LIN {X 0,Y 207.14,Z 939.529,A -85,B 0,C 180,E1 3943.742,E2 3943.742} C_VEL
LIN {X 0,Y 198.487,Z 955.966,A -85,B 0,C 180,E1 3942.665,E2 3942.665} C_VEL
LIN {X 0,Y 188.51,Z 971.483,A -85,B 0,C 180,E1 3941.219,E2 3941.219} C_VEL
LIN {X 0,Y 181.932,Z 980.299,A -85,B 0,C 180,E1 3940.126,E2 3940.126} C_VEL
LIN {X 0,Y 176.912,Z 986.053,A -85,B 0,C 180,E1 3939.583,E2 3939.583} C_VEL
LIN {X 0,Y 163.761,Z 998.092,A -85,B 0,C 180,E1 3939.087,E2 3939.087} C_VEL
LIN {X 0,Y 158.072,Z 1003.016,A -85,B 0,C 180,E1 3938.449,E2 3938.449} C_VEL
LIN {X 0,Y 156.561,Z 1004.358,A -85,B 0,C 180,E1 3938.141,E2 3938.141} C_VEL
LIN {X 0,Y 143.715,Z 1015.358,A -85,B 0,C 180,E1 3934.746,E2 3934.746} C_VEL
LIN {X 0,Y 130.308,Z 1025.353,A -85,B 0,C 180,E1 3930.116,E2 3930.116} C_VEL
LIN {X 0,Y 117.407,Z 1033.723,A -85,B 0,C 180,E1 3924,E2 3924} C_VEL
LIN {X 0,Y 106.333,Z 1040.15,A -85,B 0,C 180,E1 3916.387,E2 3916.387} C_VEL
LIN {X 0,Y 97.29,Z 1045.033,A -85,B 0,C 180,E1 3906.587,E2 3906.587} C_VEL
LIN {X 0,Y 91.724,Z 1048.097,A -85,B 0,C 180,E1 3895.157,E2 3895.157} C_VEL
LIN {X 0,Y 90.099,Z 1049.373,A -85,B 0,C 180,E1 3882.822,E2 3882.822} C_VEL
LIN {X 0,Y 91.754,Z 1048.914,A -85,B 0,C 180,E1 3871.872,E2 3871.872} C_VEL
LIN {X 0,Y 92.174,Z 1048.688,A -85,B 0,C 180,E1 3869.998,E2 3869.998} C_VEL
LIN {X 0,Y 90.722,Z 1045.5,A -85,B 0,C 180,E1 3859.842,E2 3859.842} C_VEL
LIN {X 0,Y 91.315,Z 1042.059,A -85,B 0,C 180,E1 3851.484,E2 3851.484} C_VEL
LIN {X 0,Y 94.601,Z 1042.585,A -85,B 0,C 180,E1 3838.807,E2 3838.807} C_VEL
LIN {X 0,Y 102.981,Z 1041.2,A -85,B 0,C 180,E1 3827.182,E2 3827.182} C_VEL
LIN {X 0,Y 114.76,Z 1038.132,A -85,B 0,C 180,E1 3818.213,E2 3818.213} C_VEL
LIN {X 0,Y 128.946,Z 1033.447,A -85,B 0,C 180,E1 3811.464,E2 3811.464} C_VEL
LIN {X 0,Y 142.861,Z 1028.016,A -85,B 0,C 180,E1 3806.958,E2 3806.958} C_VEL
LIN {X 0,Y 130.089,Z 1030.018,A -85,B 0,C 180,E1 3802.123,E2 3802.123} C_VEL
LIN {X 0,Y 117.737,Z 1030.209,A -85,B 0,C 180,E1 3795.768,E2 3795.768} C_VEL
LIN {X 0,Y 107.836,Z 1028.587,A -85,B 0,C 180,E1 3788.53,E2 3788.53} C_VEL
LIN {X 0,Y 99.584,Z 1024.866,A -85,B 0,C 180,E1 3779.424,E2 3779.424} C_VEL
LIN {X 0,Y 94.46,Z 1019.527,A -85,B 0,C 180,E1 3769.876,E2 3769.876} C_VEL
LIN {X 0,Y 91.911,Z 1012.221,A -85,B 0,C 180,E1 3759.627,E2 3759.627} C_VEL
LIN {X 0,Y 91.679,Z 1004.049,A -85,B 0,C 180,E1 3750.607,E2 3750.607} C_VEL
LIN {X 0,Y 93.237,Z 993.607,A -85,B 0,C 180,E1 3741.524,E2 3741.524} C_VEL
LIN {X 0,Y 95.373,Z 985.119,A -85,B 0,C 180,E1 3735.378,E2 3735.378} C_VEL
LIN {X 0,Y 97.55,Z 984.863,A -85,B 0,C 180,E1 3732.439,E2 3732.439} C_VEL
LIN {X 0,Y 100.039,Z 984.278,A -85,B 0,C 180,E1 3730.517,E2 3730.517} C_VEL
LIN {X 0,Y 103.465,Z 983.965,A -85,B 0,C 180,E1 3727.585,E2 3727.585} C_VEL
LIN {X 0,Y 106.11,Z 983.483,A -85,B 0,C 180,E1 3725.867,E2 3725.867} C_VEL
LIN {X 0,Y 110.9,Z 982.693,A -85,B 0,C 180,E1 3723.018,E2 3723.018} C_VEL
LIN {X 0,Y 118.293,Z 981.361,A -85,B 0,C 180,E1 3719.47,E2 3719.47} C_VEL
LIN {X 0,Y 120.142,Z 980.967,A -85,B 0,C 180,E1 3718.741,E2 3718.741} C_VEL
LIN {X 0,Y 112.253,Z 991.51,A -85,B 0,C 180,E1 3713.075,E2 3713.075} C_VEL
LIN {X 0,Y 104.884,Z 1000.824,A -85,B 0,C 180,E1 3706.05,E2 3706.05} C_VEL
LIN {X 0,Y 98.718,Z 1008.666,A -85,B 0,C 180,E1 3697.568,E2 3697.568} C_VEL
LIN {X 0,Y 94.402,Z 1015.031,A -85,B 0,C 180,E1 3687.573,E2 3687.573} C_VEL
LIN {X 0,Y 92.584,Z 1019.589,A -85,B 0,C 180,E1 3676.894,E2 3676.894} C_VEL
LIN {X 0,Y 93.405,Z 1022.419,A -85,B 0,C 180,E1 3666,E2 3666} C_VEL
LIN {X 0,Y 96.968,Z 1023.539,A -85,B 0,C 180,E1 3655.453,E2 3655.453} C_VEL
LIN {X 0,Y 103.213,Z 1022.966,A -85,B 0,C 180,E1 3645.776,E2 3645.776} C_VEL
LIN {X 0,Y 111.857,Z 1020.637,A -85,B 0,C 180,E1 3637.295,E2 3637.295} C_VEL
LIN {X 0,Y 122.487,Z 1016.449,A -85,B 0,C 180,E1 3630.088,E2 3630.088} C_VEL
LIN {X 0,Y 133.914,Z 1010.597,A -85,B 0,C 180,E1 3624.372,E2 3624.372} C_VEL
LIN {X 0,Y 145.608,Z 1003.273,A -85,B 0,C 180,E1 3619.825,E2 3619.825} C_VEL
LIN {X 0,Y 158.047,Z 993.888,A -85,B 0,C 180,E1 3615.932,E2 3615.932} C_VEL
LIN {X 0,Y 169.51,Z 983.568,A -85,B 0,C 180,E1 3612.953,E2 3612.953} C_VEL
LIN {X 0,Y 180.948,Z 971.298,A -85,B 0,C 180,E1 3610.405,E2 3610.405} C_VEL
LIN {X 0,Y 191.03,Z 958.248,A -85,B 0,C 180,E1 3608.419,E2 3608.419} C_VEL
LIN {X 0,Y 200.358,Z 943.599,A -85,B 0,C 180,E1 3606.749,E2 3606.749} C_VEL
LIN {X 0,Y 208.396,Z 927.988,A -85,B 0,C 180,E1 3605.407,E2 3605.407} C_VEL
LIN {X 0,Y 214.864,Z 911.992,A -85,B 0,C 180,E1 3604.36,E2 3604.36} C_VEL
LIN {X 0,Y 220.066,Z 894.686,A -85,B 0,C 180,E1 3603.504,E2 3603.504} C_VEL
LIN {X 0,Y 223.579,Z 876.803,A -85,B 0,C 180,E1 3602.869,E2 3602.869} C_VEL
LIN {X 0,Y 229.364,Z 828.556,A -85,B 0,C 180,E1 3601.817,E2 3601.817} C_VEL
LIN {X 0,Y 228.68,Z 825.976,A -85,B 0,C 180,E1 3598.998,E2 3598.998} C_VEL
LIN {X 0,Y 228.398,Z 824.641,A -85,B 0,C 180,E1 3595.481,E2 3595.481} C_VEL
LIN {X 0,Y 228.531,Z 825.221,A -85,B 0,C 180,E1 3592.964,E2 3592.964} C_VEL
LIN {X 0,Y 229.196,Z 827.412,A -85,B 0,C 180,E1 3589.824,E2 3589.824} C_VEL
LIN {X 0,Y 229.508,Z 828.787,A -85,B 0,C 180,E1 3588.784,E2 3588.784} C_VEL
LIN {X 0,Y 222.463,Z 886.283,A -85,B 0,C 180,E1 3587.683,E2 3587.683} C_VEL
LIN {X 0,Y 218.345,Z 904.811,A -85,B 0,C 180,E1 3587.221,E2 3587.221} C_VEL
LIN {X 0,Y 212.708,Z 922.213,A -85,B 0,C 180,E1 3586.66,E2 3586.66} C_VEL
LIN {X 0,Y 205.625,Z 938.773,A -85,B 0,C 180,E1 3585.946,E2 3585.946} C_VEL
LIN {X 0,Y 196.716,Z 955.353,A -85,B 0,C 180,E1 3584.953,E2 3584.953} C_VEL
LIN {X 0,Y 186.536,Z 970.767,A -85,B 0,C 180,E1 3583.628,E2 3583.628} C_VEL
LIN {X 0,Y 175.18,Z 985.129,A -85,B 0,C 180,E1 3581.861,E2 3581.861} C_VEL
LIN {X 0,Y 162.615,Z 998.588,A -85,B 0,C 180,E1 3579.484,E2 3579.484} C_VEL
LIN {X 0,Y 156.561,Z 1004.358,A -85,B 0,C 180,E1 3578.141,E2 3578.141} C_VEL
LIN {X 0,Y 150.863,Z 1009.035,A -85,B 0,C 180,E1 3577.195,E2 3577.195} C_VEL
LIN {X 0,Y 136.124,Z 1018.528,A -85,B 0,C 180,E1 3575.726,E2 3575.726} C_VEL
LIN {X 0,Y 129.953,Z 1022.27,A -85,B 0,C 180,E1 3574.524,E2 3574.524} C_VEL
LIN {X 0,Y 128.362,Z 1023.303,A -85,B 0,C 180,E1 3574.028,E2 3574.028} C_VEL
LIN {X 0,Y 114.948,Z 1031.623,A -85,B 0,C 180,E1 3568.476,E2 3568.476} C_VEL
LIN {X 0,Y 102.675,Z 1038.276,A -85,B 0,C 180,E1 3561.171,E2 3561.171} C_VEL
LIN {X 0,Y 92.183,Z 1043.336,A -85,B 0,C 180,E1 3551.423,E2 3551.423} C_VEL
LIN {X 0,Y 85.11,Z 1046.569,A -85,B 0,C 180,E1 3539.563,E2 3539.563} C_VEL
LIN {X 0,Y 82.202,Z 1048.054,A -85,B 0,C 180,E1 3525.519,E2 3525.519} C_VEL
LIN {X 0,Y 83.579,Z 1047.647,A -85,B 0,C 180,E1 3512.741,E2 3512.741} C_VEL
LIN {X 0,Y 84.182,Z 1047.32,A -85,B 0,C 180,E1 3509.998,E2 3509.998} C_VEL
LIN {X 0,Y 82.765,Z 1044.032,A -85,B 0,C 180,E1 3498.853,E2 3498.853} C_VEL
LIN {X 0,Y 83.874,Z 1039.964,A -85,B 0,C 180,E1 3489.043,E2 3489.043} C_VEL
LIN {X 0,Y 88.472,Z 1040.751,A -85,B 0,C 180,E1 3474.802,E2 3474.802} C_VEL
LIN {X 0,Y 98.105,Z 1039.658,A -85,B 0,C 180,E1 3463.065,E2 3463.065} C_VEL
LIN {X 0,Y 111.2,Z 1036.873,A -85,B 0,C 180,E1 3454.183,E2 3454.183} C_VEL
LIN {X 0,Y 126.523,Z 1032.56,A -85,B 0,C 180,E1 3447.735,E2 3447.735} C_VEL
LIN {X 0,Y 129.706,Z 1031.51,A -85,B 0,C 180,E1 3446.59,E2 3446.59} C_VEL
LIN {X 0,Y 116.781,Z 1031.94,A -85,B 0,C 180,E1 3441.051,E2 3441.051} C_VEL
LIN {X 0,Y 104.822,Z 1030.492,A -85,B 0,C 180,E1 3433.795,E2 3433.795} C_VEL
LIN {X 0,Y 95.389,Z 1027.21,A -85,B 0,C 180,E1 3425.245,E2 3425.245} C_VEL
LIN {X 0,Y 88.329,Z 1021.868,A -85,B 0,C 180,E1 3414.803,E2 3414.803} C_VEL
LIN {X 0,Y 84.65,Z 1015.06,A -85,B 0,C 180,E1 3404.235,E2 3404.235} C_VEL
LIN {X 0,Y 83.566,Z 1006.738,A -85,B 0,C 180,E1 3393.722,E2 3393.722} C_VEL
LIN {X 0,Y 84.614,Z 996.726,A -85,B 0,C 180,E1 3383.782,E2 3383.782} C_VEL
LIN {X 0,Y 85.944,Z 990.841,A -85,B 0,C 180,E1 3378.682,E2 3378.682} C_VEL
LIN {X 0,Y 87.93,Z 990.529,A -85,B 0,C 180,E1 3375.168,E2 3375.168} C_VEL
LIN {X 0,Y 90.155,Z 990.042,A -85,B 0,C 180,E1 3372.946,E2 3372.946} C_VEL
LIN {X 0,Y 93.358,Z 989.753,A -85,B 0,C 180,E1 3369.544,E2 3369.544} C_VEL
LIN {X 0,Y 95.811,Z 989.38,A -85,B 0,C 180,E1 3367.521,E2 3367.521} C_VEL
LIN {X 0,Y 106.784,Z 987.714,A -85,B 0,C 180,E1 3360.52,E2 3360.52} C_VEL
LIN {X 0,Y 110.219,Z 987.236,A -85,B 0,C 180,E1 3358.739,E2 3358.739} C_VEL
LIN {X 0,Y 101.656,Z 997.624,A -85,B 0,C 180,E1 3351.949,E2 3351.949} C_VEL
LIN {X 0,Y 94.103,Z 1006.401,A -85,B 0,C 180,E1 3343.52,E2 3343.52} C_VEL
LIN {X 0,Y 88.303,Z 1013.637,A -85,B 0,C 180,E1 3333.247,E2 3333.247} C_VEL
LIN {X 0,Y 85.137,Z 1018.99,A -85,B 0,C 180,E1 3321.9,E2 3321.9} C_VEL
LIN {X 0,Y 84.842,Z 1022.57,A -85,B 0,C 180,E1 3310.018,E2 3310.018} C_VEL
LIN {X 0,Y 87.558,Z 1024.448,A -85,B 0,C 180,E1 3298.314,E2 3298.314} C_VEL
LIN {X 0,Y 93.679,Z 1024.614,A -85,B 0,C 180,E1 3286.917,E2 3286.917} C_VEL
LIN {X 0,Y 102.199,Z 1023.005,A -85,B 0,C 180,E1 3277.586,E2 3277.586} C_VEL
LIN {X 0,Y 112.979,Z 1019.537,A -85,B 0,C 180,E1 3269.71,E2 3269.71} C_VEL
LIN {X 0,Y 124.456,Z 1014.517,A -85,B 0,C 180,E1 3263.675,E2 3263.675} C_VEL
LIN {X 0,Y 137.154,Z 1007.544,A -85,B 0,C 180,E1 3258.614,E2 3258.614} C_VEL
LIN {X 0,Y 149.837,Z 999.035,A -85,B 0,C 180,E1 3254.633,E2 3254.633} C_VEL
LIN {X 0,Y 162.208,Z 989.045,A -85,B 0,C 180,E1 3251.458,E2 3251.458} C_VEL
LIN {X 0,Y 174.061,Z 977.537,A -85,B 0,C 180,E1 3248.883,E2 3248.883} C_VEL
LIN {X 0,Y 184.856,Z 964.933,A -85,B 0,C 180,E1 3246.835,E2 3246.835} C_VEL
LIN {X 0,Y 194.755,Z 951,A -85,B 0,C 180,E1 3245.146,E2 3245.146} C_VEL
LIN {X 0,Y 203.413,Z 936.091,A -85,B 0,C 180,E1 3243.784,E2 3243.784} C_VEL
LIN {X 0,Y 210.7,Z 920.386,A -85,B 0,C 180,E1 3242.689,E2 3242.689} C_VEL
LIN {X 0,Y 216.526,Z 904.044,A -85,B 0,C 180,E1 3241.818,E2 3241.818} C_VEL
LIN {X 0,Y 220.977,Z 886.41,A -85,B 0,C 180,E1 3241.116,E2 3241.116} C_VEL
LIN {X 0,Y 223.926,Z 866.992,A -85,B 0,C 180,E1 3240.57,E2 3240.57} C_VEL
LIN {X 0,Y 227.81,Z 834.873,A -85,B 0,C 180,E1 3239.938,E2 3239.938} C_VEL
LIN {X 0,Y 227.542,Z 833.599,A -85,B 0,C 180,E1 3238.238,E2 3238.238} C_VEL
LIN {X 0,Y 227.394,Z 832.579,A -85,B 0,C 180,E1 3235.461,E2 3235.461} C_VEL
LIN {X 0,Y 227.497,Z 833.107,A -85,B 0,C 180,E1 3233.185,E2 3233.185} C_VEL
LIN {X 0,Y 227.918,Z 834.797,A -85,B 0,C 180,E1 3230.672,E2 3230.672} C_VEL
LIN {X 0,Y 221.505,Z 885.672,A -85,B 0,C 180,E1 3229.745,E2 3229.745} C_VEL
LIN {X 0,Y 217.294,Z 904.226,A -85,B 0,C 180,E1 3229.32,E2 3229.32} C_VEL
LIN {X 0,Y 211.491,Z 921.79,A -85,B 0,C 180,E1 3228.807,E2 3228.807} C_VEL
LIN {X 0,Y 204.311,Z 938.243,A -85,B 0,C 180,E1 3228.168,E2 3228.168} C_VEL
LIN {X 0,Y 195.301,Z 954.667,A -85,B 0,C 180,E1 3227.283,E2 3227.283} C_VEL
LIN {X 0,Y 184.9,Z 970.051,A -85,B 0,C 180,E1 3226.083,E2 3226.083} C_VEL
LIN {X 0,Y 173.298,Z 984.353,A -85,B 0,C 180,E1 3224.474,E2 3224.474} C_VEL
LIN {X 0,Y 160.56,Z 997.605,A -85,B 0,C 180,E1 3222.319,E2 3222.319} C_VEL
LIN {X 0,Y 147.301,Z 1009.351,A -85,B 0,C 180,E1 3219.506,E2 3219.506} C_VEL
LIN {X 0,Y 133.73,Z 1019.663,A -85,B 0,C 180,E1 3215.802,E2 3215.802} C_VEL
LIN {X 0,Y 128.362,Z 1023.303,A -85,B 0,C 180,E1 3214.028,E2 3214.028} C_VEL
LIN {X 0,Y 122.39,Z 1026.785,A -85,B 0,C 180,E1 3212.393,E2 3212.393} C_VEL
LIN {X 0,Y 106.111,Z 1033.73,A -85,B 0,C 180,E1 3208.868,E2 3208.868} C_VEL
LIN {X 0,Y 100.166,Z 1036.16,A -85,B 0,C 180,E1 3206.473,E2 3206.473} C_VEL
LIN {X 0,Y 99.437,Z 1036.509,A -85,B 0,C 180,E1 3206.04,E2 3206.04} C_VEL
LIN {X 0,Y 87.809,Z 1041.638,A -85,B 0,C 180,E1 3196.78,E2 3196.78} C_VEL
LIN {X 0,Y 79.076,Z 1045.041,A -85,B 0,C 180,E1 3184.678,E2 3184.678} C_VEL
LIN {X 0,Y 74.685,Z 1046.669,A -85,B 0,C 180,E1 3170.368,E2 3170.368} C_VEL
LIN {X 0,Y 75.097,Z 1046.49,A -85,B 0,C 180,E1 3155.346,E2 3155.346} C_VEL
LIN {X 0,Y 76.178,Z 1045.929,A -85,B 0,C 180,E1 3149.998,E2 3149.998} C_VEL
LIN {X 0,Y 74.85,Z 1042.348,A -85,B 0,C 180,E1 3137.192,E2 3137.192} C_VEL
LIN {X 0,Y 76.757,Z 1037.873,A -85,B 0,C 180,E1 3125.363,E2 3125.363} C_VEL
LIN {X 0,Y 82.436,Z 1038.835,A -85,B 0,C 180,E1 3110.895,E2 3110.895} C_VEL
LIN {X 0,Y 93.574,Z 1038.059,A -85,B 0,C 180,E1 3098.735,E2 3098.735} C_VEL
LIN {X 0,Y 108.374,Z 1035.586,A -85,B 0,C 180,E1 3089.857,E2 3089.857} C_VEL
LIN {X 0,Y 116.86,Z 1033.639,A -85,B 0,C 180,E1 3086.333,E2 3086.333} C_VEL
LIN {X 0,Y 104.261,Z 1032.609,A -85,B 0,C 180,E1 3080.195,E2 3080.195} C_VEL
LIN {X 0,Y 92.615,Z 1029.612,A -85,B 0,C 180,E1 3071.835,E2 3071.835} C_VEL
LIN {X 0,Y 83.98,Z 1024.926,A -85,B 0,C 180,E1 3062.046,E2 3062.046} C_VEL
LIN {X 0,Y 78.132,Z 1018.14,A -85,B 0,C 180,E1 3050.2,E2 3050.2} C_VEL
LIN {X 0,Y 75.824,Z 1010.508,A -85,B 0,C 180,E1 3039.141,E2 3039.141} C_VEL
LIN {X 0,Y 75.889,Z 1001.295,A -85,B 0,C 180,E1 3028.195,E2 3028.195} C_VEL
LIN {X 0,Y 76.723,Z 996.268,A -85,B 0,C 180,E1 3022.869,E2 3022.869} C_VEL
LIN {X 0,Y 78.515,Z 995.876,A -85,B 0,C 180,E1 3018.53,E2 3018.53} C_VEL
LIN {X 0,Y 80.45,Z 995.483,A -85,B 0,C 180,E1 3015.892,E2 3015.892} C_VEL
LIN {X 0,Y 83.379,Z 995.174,A -85,B 0,C 180,E1 3011.968,E2 3011.968} C_VEL
LIN {X 0,Y 85.609,Z 994.889,A -85,B 0,C 180,E1 3009.568,E2 3009.568} C_VEL
LIN {X 0,Y 95.363,Z 993.556,A -85,B 0,C 180,E1 3001.865,E2 3001.865} C_VEL
LIN {X 0,Y 100.299,Z 992.999,A -85,B 0,C 180,E1 2998.776,E2 2998.776} C_VEL
LIN {X 0,Y 91.562,Z 1002.649,A -85,B 0,C 180,E1 2991.124,E2 2991.124} C_VEL
LIN {X 0,Y 84.22,Z 1010.6,A -85,B 0,C 180,E1 2981.646,E2 2981.646} C_VEL
LIN {X 0,Y 78.96,Z 1017.066,A -85,B 0,C 180,E1 2970.002,E2 2970.002} C_VEL
LIN {X 0,Y 76.727,Z 1021.728,A -85,B 0,C 180,E1 2957.203,E2 2957.203} C_VEL
LIN {X 0,Y 77.798,Z 1024.694,A -85,B 0,C 180,E1 2944.091,E2 2944.091} C_VEL
LIN {X 0,Y 82.241,Z 1025.963,A -85,B 0,C 180,E1 2931.683,E2 2931.683} C_VEL
LIN {X 0,Y 89.783,Z 1025.523,A -85,B 0,C 180,E1 2920.778,E2 2920.778} C_VEL
LIN {X 0,Y 99.888,Z 1023.34,A -85,B 0,C 180,E1 2911.7,E2 2911.7} C_VEL
LIN {X 0,Y 111.944,Z 1019.322,A -85,B 0,C 180,E1 2904.354,E2 2904.354} C_VEL
LIN {X 0,Y 124.784,Z 1013.631,A -85,B 0,C 180,E1 2898.695,E2 2898.695} C_VEL
LIN {X 0,Y 138.192,Z 1006.076,A -85,B 0,C 180,E1 2894.184,E2 2894.184} C_VEL
LIN {X 0,Y 151.57,Z 996.816,A -85,B 0,C 180,E1 2890.614,E2 2890.614} C_VEL
LIN {X 0,Y 164.488,Z 985.99,A -85,B 0,C 180,E1 2887.778,E2 2887.778} C_VEL
LIN {X 0,Y 176.782,Z 973.55,A -85,B 0,C 180,E1 2885.485,E2 2885.485} C_VEL
LIN {X 0,Y 187.872,Z 959.849,A -85,B 0,C 180,E1 2883.662,E2 2883.662} C_VEL
LIN {X 0,Y 197.617,Z 945.175,A -85,B 0,C 180,E1 2882.21,E2 2882.21} C_VEL
LIN {X 0,Y 206.003,Z 929.533,A -85,B 0,C 180,E1 2881.04,E2 2881.04} C_VEL
LIN {X 0,Y 212.968,Z 912.92,A -85,B 0,C 180,E1 2880.094,E2 2880.094} C_VEL
LIN {X 0,Y 218.294,Z 895.647,A -85,B 0,C 180,E1 2879.347,E2 2879.347} C_VEL
LIN {X 0,Y 221.909,Z 877.803,A -85,B 0,C 180,E1 2878.782,E2 2878.782} C_VEL
LIN {X 0,Y 226.502,Z 841.495,A -85,B 0,C 180,E1 2878.044,E2 2878.044} C_VEL
LIN {X 0,Y 226.39,Z 840.516,A -85,B 0,C 180,E1 2875.441,E2 2875.441} C_VEL
LIN {X 0,Y 226.466,Z 840.998,A -85,B 0,C 180,E1 2873.401,E2 2873.401} C_VEL
LIN {X 0,Y 226.514,Z 841.714,A -85,B 0,C 180,E1 2872.569,E2 2872.569} C_VEL
LIN {X 0,Y 220.863,Z 885,A -85,B 0,C 180,E1 2871.825,E2 2871.825} C_VEL
LIN {X 0,Y 216.537,Z 903.642,A -85,B 0,C 180,E1 2871.438,E2 2871.438} C_VEL
LIN {X 0,Y 210.574,Z 921.366,A -85,B 0,C 180,E1 2870.977,E2 2870.977} C_VEL
LIN {X 0,Y 202.824,Z 938.71,A -85,B 0,C 180,E1 2870.376,E2 2870.376} C_VEL
LIN {X 0,Y 193.598,Z 954.919,A -85,B 0,C 180,E1 2869.586,E2 2869.586} C_VEL
LIN {X 0,Y 183.133,Z 969.949,A -85,B 0,C 180,E1 2868.525,E2 2868.525} C_VEL
LIN {X 0,Y 170.845,Z 984.61,A -85,B 0,C 180,E1 2867.011,E2 2867.011} C_VEL
LIN {X 0,Y 158.289,Z 997.209,A -85,B 0,C 180,E1 2865.114,E2 2865.114} C_VEL
LIN {X 0,Y 144.653,Z 1008.83,A -85,B 0,C 180,E1 2862.526,E2 2862.526} C_VEL
LIN {X 0,Y 130.595,Z 1019.011,A -85,B 0,C 180,E1 2859.073,E2 2859.073} C_VEL
LIN {X 0,Y 116.413,Z 1027.718,A -85,B 0,C 180,E1 2854.398,E2 2854.398} C_VEL
LIN {X 0,Y 102.63,Z 1034.956,A -85,B 0,C 180,E1 2847.948,E2 2847.948} C_VEL
LIN {X 0,Y 99.437,Z 1036.509,A -85,B 0,C 180,E1 2846.04,E2 2846.04} C_VEL
LIN {X 0,Y 93.849,Z 1038.723,A -85,B 0,C 180,E1 2843.117,E2 2843.117} C_VEL
LIN {X 0,Y 79.687,Z 1042.18,A -85,B 0,C 180,E1 2836.214,E2 2836.214} C_VEL
LIN {X 0,Y 74.402,Z 1043.332,A -85,B 0,C 180,E1 2831.492,E2 2831.492} C_VEL
LIN {X 0,Y 73.625,Z 1043.541,A -85,B 0,C 180,E1 2830.362,E2 2830.362} C_VEL
LIN {X 0,Y 67.399,Z 1045.341,A -85,B 0,C 180,E1 2814.541,E2 2814.541} C_VEL
LIN {X 0,Y 66.807,Z 1045.257,A -85,B 0,C 180,E1 2797.739,E2 2797.739} C_VEL
LIN {X 0,Y 68.157,Z 1044.534,A -85,B 0,C 180,E1 2789.998,E2 2789.998} C_VEL
LIN {X 0,Y 66.998,Z 1040.713,A -85,B 0,C 180,E1 2775.301,E2 2775.301} C_VEL
LIN {X 0,Y 69.833,Z 1035.594,A -85,B 0,C 180,E1 2761.801,E2 2761.801} C_VEL
LIN {X 0,Y 77.357,Z 1036.853,A -85,B 0,C 180,E1 2745.733,E2 2745.733} C_VEL
LIN {X 0,Y 90.12,Z 1036.353,A -85,B 0,C 180,E1 2733.681,E2 2733.681} C_VEL
LIN {X 0,Y 104.045,Z 1034.516,A -85,B 0,C 180,E1 2726.081,E2 2726.081} C_VEL
LIN {X 0,Y 91.69,Z 1032.057,A -85,B 0,C 180,E1 2719.094,E2 2719.094} C_VEL
LIN {X 0,Y 80.514,Z 1027.507,A -85,B 0,C 180,E1 2709.289,E2 2709.289} C_VEL
LIN {X 0,Y 72.768,Z 1021.263,A -85,B 0,C 180,E1 2697.636,E2 2697.636} C_VEL
LIN {X 0,Y 68.519,Z 1013.201,A -85,B 0,C 180,E1 2684.395,E2 2684.395} C_VEL
LIN {X 0,Y 67.646,Z 1003.97,A -85,B 0,C 180,E1 2671.77,E2 2671.77} C_VEL
LIN {X 0,Y 67.887,Z 1001.313,A -85,B 0,C 180,E1 2667.978,E2 2667.978} C_VEL
LIN {X 0,Y 69.42,Z 1001.045,A -85,B 0,C 180,E1 2662.775,E2 2662.775} C_VEL
LIN {X 0,Y 70.682,Z 1000.717,A -85,B 0,C 180,E1 2660.462,E2 2660.462} C_VEL
LIN {X 0,Y 73.602,Z 1000.334,A -85,B 0,C 180,E1 2655.055,E2 2655.055} C_VEL
LIN {X 0,Y 84.038,Z 998.963,A -85,B 0,C 180,E1 2643.606,E2 2643.606} C_VEL
LIN {X 0,Y 90.469,Z 998.2,A -85,B 0,C 180,E1 2638.936,E2 2638.936} C_VEL
LIN {X 0,Y 81.442,Z 1007.282,A -85,B 0,C 180,E1 2630.108,E2 2630.108} C_VEL
LIN {X 0,Y 74.387,Z 1014.48,A -85,B 0,C 180,E1 2619.284,E2 2619.284} C_VEL
LIN {X 0,Y 69.837,Z 1020.219,A -85,B 0,C 180,E1 2605.897,E2 2605.897} C_VEL
LIN {X 0,Y 68.842,Z 1024.218,A -85,B 0,C 180,E1 2591.368,E2 2591.368} C_VEL
LIN {X 0,Y 71.768,Z 1026.594,A -85,B 0,C 180,E1 2576.713,E2 2576.713} C_VEL
LIN {X 0,Y 78.6,Z 1027.221,A -85,B 0,C 180,E1 2563.526,E2 2563.526} C_VEL
LIN {X 0,Y 88.474,Z 1025.992,A -85,B 0,C 180,E1 2552.853,E2 2552.853} C_VEL
LIN {X 0,Y 100.924,Z 1022.847,A -85,B 0,C 180,E1 2544.297,E2 2544.297} C_VEL
LIN {X 0,Y 113.676,Z 1018.229,A -85,B 0,C 180,E1 2538.21,E2 2538.21} C_VEL
LIN {X 0,Y 127.42,Z 1011.773,A -85,B 0,C 180,E1 2533.344,E2 2533.344} C_VEL
LIN {X 0,Y 140.96,Z 1003.779,A -85,B 0,C 180,E1 2529.619,E2 2529.619} C_VEL
LIN {X 0,Y 154.03,Z 994.346,A -85,B 0,C 180,E1 2526.707,E2 2526.707} C_VEL
LIN {X 0,Y 166.727,Z 983.294,A -85,B 0,C 180,E1 2524.336,E2 2524.336} C_VEL
LIN {X 0,Y 178.632,Z 970.822,A -85,B 0,C 180,E1 2522.421,E2 2522.421} C_VEL
LIN {X 0,Y 189.443,Z 957.126,A -85,B 0,C 180,E1 2520.872,E2 2520.872} C_VEL
LIN {X 0,Y 198.974,Z 942.355,A -85,B 0,C 180,E1 2519.621,E2 2519.621} C_VEL
LIN {X 0,Y 207.029,Z 926.703,A -85,B 0,C 180,E1 2518.614,E2 2518.614} C_VEL
LIN {X 0,Y 213.625,Z 910.169,A -85,B 0,C 180,E1 2517.795,E2 2517.795} C_VEL
LIN {X 0,Y 218.814,Z 892.219,A -85,B 0,C 180,E1 2517.119,E2 2517.119} C_VEL
LIN {X 0,Y 222.109,Z 874.388,A -85,B 0,C 180,E1 2516.625,E2 2516.625} C_VEL
LIN {X 0,Y 225.387,Z 848.568,A -85,B 0,C 180,E1 2516.121,E2 2516.121} C_VEL
LIN {X 0,Y 225.381,Z 848.716,A -85,B 0,C 180,E1 2514.487,E2 2514.487} C_VEL
LIN {X 0,Y 220.502,Z 884.714,A -85,B 0,C 180,E1 2513.908,E2 2513.908} C_VEL
LIN {X 0,Y 215.958,Z 903.747,A -85,B 0,C 180,E1 2513.554,E2 2513.554} C_VEL
LIN {X 0,Y 209.779,Z 921.573,A -85,B 0,C 180,E1 2513.147,E2 2513.147} C_VEL
LIN {X 0,Y 202.132,Z 938.23,A -85,B 0,C 180,E1 2512.647,E2 2512.647} C_VEL
LIN {X 0,Y 192.858,Z 954.202,A -85,B 0,C 180,E1 2511.977,E2 2511.977} C_VEL
LIN {X 0,Y 182.188,Z 969.235,A -85,B 0,C 180,E1 2511.055,E2 2511.055} C_VEL
LIN {X 0,Y 169.693,Z 983.838,A -85,B 0,C 180,E1 2509.73,E2 2509.73} C_VEL
LIN {X 0,Y 156.404,Z 996.814,A -85,B 0,C 180,E1 2507.981,E2 2507.981} C_VEL
LIN {X 0,Y 142.422,Z 1008.3,A -85,B 0,C 180,E1 2505.649,E2 2505.649} C_VEL
LIN {X 0,Y 127.905,Z 1018.319,A -85,B 0,C 180,E1 2502.493,E2 2502.493} C_VEL
LIN {X 0,Y 113.114,Z 1026.915,A -85,B 0,C 180,E1 2498.143,E2 2498.143} C_VEL
LIN {X 0,Y 98.514,Z 1034.047,A -85,B 0,C 180,E1 2492.003,E2 2492.003} C_VEL
LIN {X 0,Y 84.928,Z 1039.621,A -85,B 0,C 180,E1 2483.181,E2 2483.181} C_VEL
LIN {X 0,Y 74.224,Z 1043.342,A -85,B 0,C 180,E1 2471.303,E2 2471.303} C_VEL
LIN {X 0,Y 73.625,Z 1043.541,A -85,B 0,C 180,E1 2470.362,E2 2470.362} C_VEL
LIN {X 0,Y 69.727,Z 1044.333,A -85,B 0,C 180,E1 2465.015,E2 2465.015} C_VEL
LIN {X 0,Y 60.453,Z 1044.534,A -85,B 0,C 180,E1 2451.447,E2 2451.447} C_VEL
LIN {X 0,Y 58.557,Z 1044.173,A -85,B 0,C 180,E1 2443.613,E2 2443.613} C_VEL
LIN {X 0,Y 58.558,Z 1044.082,A -85,B 0,C 180,E1 2441.98,E2 2441.98} C_VEL
LIN {X 0,Y 60.12,Z 1043.139,A -85,B 0,C 180,E1 2429.997,E2 2429.997} C_VEL
LIN {X 0,Y 59.204,Z 1039.198,A -85,B 0,C 180,E1 2413.313,E2 2413.313} C_VEL
LIN {X 0,Y 63.606,Z 1033.321,A -85,B 0,C 180,E1 2396.42,E2 2396.42} C_VEL
LIN {X 0,Y 73.019,Z 1034.774,A -85,B 0,C 180,E1 2379.928,E2 2379.928} C_VEL
LIN {X 0,Y 87.438,Z 1034.543,A -85,B 0,C 180,E1 2368.294,E2 2368.294} C_VEL
LIN {X 0,Y 91.483,Z 1034.201,A -85,B 0,C 180,E1 2365.923,E2 2365.923} C_VEL
LIN {X 0,Y 79.145,Z 1030.264,A -85,B 0,C 180,E1 2357.648,E2 2357.648} C_VEL
LIN {X 0,Y 68.607,Z 1024.115,A -85,B 0,C 180,E1 2345.854,E2 2345.854} C_VEL
LIN {X 0,Y 62.386,Z 1016.75,A -85,B 0,C 180,E1 2332.632,E2 2332.632} C_VEL
LIN {X 0,Y 59.773,Z 1007.923,A -85,B 0,C 180,E1 2318.405,E2 2318.405} C_VEL
LIN {X 0,Y 59.614,Z 1006.28,A -85,B 0,C 180,E1 2315.207,E2 2315.207} C_VEL
LIN {X 0,Y 60.732,Z 1005.885,A -85,B 0,C 180,E1 2308.206,E2 2308.206} C_VEL
LIN {X 0,Y 64.059,Z 1005.228,A -85,B 0,C 180,E1 2299.036,E2 2299.036} C_VEL
LIN {X 0,Y 73.521,Z 1003.896,A -85,B 0,C 180,E1 2285.313,E2 2285.313} C_VEL
LIN {X 0,Y 80.604,Z 1003.037,A -85,B 0,C 180,E1 2279.154,E2 2279.154} C_VEL
LIN {X 0,Y 71.301,Z 1011.564,A -85,B 0,C 180,E1 2268.818,E2 2268.818} C_VEL
LIN {X 0,Y 64.642,Z 1018.067,A -85,B 0,C 180,E1 2256.218,E2 2256.218} C_VEL
LIN {X 0,Y 61.07,Z 1023.132,A -85,B 0,C 180,E1 2240.579,E2 2240.579} C_VEL
LIN {X 0,Y 61.738,Z 1026.491,A -85,B 0,C 180,E1 2224.073,E2 2224.073} C_VEL
LIN {X 0,Y 67.143,Z 1028.254,A -85,B 0,C 180,E1 2207.927,E2 2207.927} C_VEL
LIN {X 0,Y 76.072,Z 1028.199,A -85,B 0,C 180,E1 2195.334,E2 2195.334} C_VEL
LIN {X 0,Y 87.623,Z 1026.411,A -85,B 0,C 180,E1 2185.653,E2 2185.653} C_VEL
LIN {X 0,Y 101.073,Z 1022.755,A -85,B 0,C 180,E1 2178.258,E2 2178.258} C_VEL
LIN {X 0,Y 114.88,Z 1017.541,A -85,B 0,C 180,E1 2172.898,E2 2172.898} C_VEL
LIN {X 0,Y 129.458,Z 1010.421,A -85,B 0,C 180,E1 2168.666,E2 2168.666} C_VEL
LIN {X 0,Y 143.627,Z 1001.785,A -85,B 0,C 180,E1 2165.452,E2 2165.452} C_VEL
LIN {X 0,Y 157.37,Z 991.499,A -85,B 0,C 180,E1 2162.914,E2 2162.914} C_VEL
LIN {X 0,Y 170.355,Z 979.618,A -85,B 0,C 180,E1 2160.887,E2 2160.887} C_VEL
LIN {X 0,Y 182.248,Z 966.43,A -85,B 0,C 180,E1 2159.269,E2 2159.269} C_VEL
LIN {X 0,Y 192.588,Z 952.496,A -85,B 0,C 180,E1 2158,E2 2158} C_VEL
LIN {X 0,Y 201.755,Z 937.309,A -85,B 0,C 180,E1 2156.952,E2 2156.952} C_VEL
LIN {X 0,Y 209.454,Z 921.22,A -85,B 0,C 180,E1 2156.098,E2 2156.098} C_VEL
LIN {X 0,Y 213.993,Z 909.105,A -85,B 0,C 180,E1 2155.585,E2 2155.585} C_VEL
LIN {X 0,Y 207.189,Z 926.575,A -85,B 0,C 180,E1 2155.222,E2 2155.222} C_VEL
LIN {X 0,Y 198.799,Z 943.193,A -85,B 0,C 180,E1 2154.765,E2 2154.765} C_VEL
LIN {X 0,Y 188.956,Z 958.812,A -85,B 0,C 180,E1 2154.147,E2 2154.147} C_VEL
LIN {X 0,Y 177.692,Z 973.4,A -85,B 0,C 180,E1 2153.285,E2 2153.285} C_VEL
LIN {X 0,Y 165.532,Z 986.546,A -85,B 0,C 180,E1 2152.133,E2 2152.133} C_VEL
LIN {X 0,Y 151.978,Z 998.862,A -85,B 0,C 180,E1 2150.534,E2 2150.534} C_VEL
LIN {X 0,Y 136.859,Z 1010.376,A -85,B 0,C 180,E1 2148.224,E2 2148.224} C_VEL
LIN {X 0,Y 122.021,Z 1019.812,A -85,B 0,C 180,E1 2145.215,E2 2145.215} C_VEL
LIN {X 0,Y 106.078,Z 1028.235,A -85,B 0,C 180,E1 2140.738,E2 2140.738} C_VEL
LIN {X 0,Y 90.885,Z 1034.777,A -85,B 0,C 180,E1 2134.434,E2 2134.434} C_VEL
LIN {X 0,Y 76.794,Z 1039.708,A -85,B 0,C 180,E1 2125.107,E2 2125.107} C_VEL
LIN {X 0,Y 65.275,Z 1042.944,A -85,B 0,C 180,E1 2111.194,E2 2111.194} C_VEL
LIN {X 0,Y 59.262,Z 1044.211,A -85,B 0,C 180,E1 2093.884,E2 2093.884} C_VEL
LIN {X 0,Y 58.558,Z 1044.082,A -85,B 0,C 180,E1 2081.98,E2 2081.98} C_VEL
LIN {X 0,Y 57.962,Z 1043.69,A -85,B 0,C 180,E1 2077.757,E2 2077.757} C_VEL
LIN {X 0,Y 55.681,Z 1042.691,A -85,B 0,C 180,E1 2072.307,E2 2072.307} C_VEL
LIN {X 0,Y 51.246,Z 1040.071,A -85,B 0,C 180,E1 2060.965,E2 2060.965} C_VEL
LIN {X 0,Y 51.039,Z 1039.532,A -85,B 0,C 180,E1 2058.409,E2 2058.409} C_VEL
LIN {X 0,Y 54.131,Z 1034.109,A -85,B 0,C 180,E1 2038.853,E2 2038.853} C_VEL
LIN {X 0,Y 57.941,Z 1030.913,A -85,B 0,C 180,E1 2030.317,E2 2030.317} C_VEL
LIN {X 0,Y 70.21,Z 1032.678,A -85,B 0,C 180,E1 2012.833,E2 2012.833} C_VEL
LIN {X 0,Y 79.349,Z 1032.819,A -85,B 0,C 180,E1 2005.987,E2 2005.987} C_VEL
LIN {X 0,Y 67.359,Z 1027.594,A -85,B 0,C 180,E1 1996.38,E2 1996.38} C_VEL
LIN {X 0,Y 57.968,Z 1020.368,A -85,B 0,C 180,E1 1982.964,E2 1982.964} C_VEL
LIN {X 0,Y 52.515,Z 1011.148,A -85,B 0,C 180,E1 1965.386,E2 1965.386} C_VEL
LIN {X 0,Y 52.481,Z 1010.622,A -85,B 0,C 180,E1 1956.414,E2 1956.414} C_VEL
LIN {X 0,Y 54.671,Z 1009.874,A -85,B 0,C 180,E1 1944.822,E2 1944.822} C_VEL
LIN {X 0,Y 57.818,Z 1009.35,A -85,B 0,C 180,E1 1936.23,E2 1936.23} C_VEL
LIN {X 0,Y 70.538,Z 1007.709,A -85,B 0,C 180,E1 1919.28,E2 1919.28} C_VEL
LIN {X 0,Y 61.148,Z 1015.546,A -85,B 0,C 180,E1 1907.12,E2 1907.12} C_VEL
LIN {X 0,Y 54.783,Z 1021.69,A -85,B 0,C 180,E1 1891.049,E2 1891.049} C_VEL
LIN {X 0,Y 52.916,Z 1026.007,A -85,B 0,C 180,E1 1872.406,E2 1872.406} C_VEL
LIN {X 0,Y 56.118,Z 1028.648,A -85,B 0,C 180,E1 1853.991,E2 1853.991} C_VEL
LIN {X 0,Y 64.481,Z 1029.648,A -85,B 0,C 180,E1 1837.741,E2 1837.741} C_VEL
LIN {X 0,Y 75.803,Z 1028.857,A -85,B 0,C 180,E1 1826.246,E2 1826.246} C_VEL
LIN {X 0,Y 89.285,Z 1026.316,A -85,B 0,C 180,E1 1817.852,E2 1817.852} C_VEL
LIN {X 0,Y 104.277,Z 1021.807,A -85,B 0,C 180,E1 1811.618,E2 1811.618} C_VEL
LIN {X 0,Y 118.947,Z 1015.823,A -85,B 0,C 180,E1 1807.245,E2 1807.245} C_VEL
LIN {X 0,Y 134.27,Z 1007.803,A -85,B 0,C 180,E1 1803.775,E2 1803.775} C_VEL
LIN {X 0,Y 148.911,Z 998.235,A -85,B 0,C 180,E1 1801.155,E2 1801.155} C_VEL
LIN {X 0,Y 162.339,Z 987.457,A -85,B 0,C 180,E1 1799.161,E2 1799.161} C_VEL
LIN {X 0,Y 175.136,Z 974.924,A -85,B 0,C 180,E1 1797.526,E2 1797.526} C_VEL
LIN {X 0,Y 185.096,Z 963.267,A -85,B 0,C 180,E1 1796.39,E2 1796.39} C_VEL
LIN {X 0,Y 173.137,Z 977.612,A -85,B 0,C 180,E1 1795.597,E2 1795.597} C_VEL
LIN {X 0,Y 159.718,Z 990.895,A -85,B 0,C 180,E1 1794.471,E2 1794.471} C_VEL
LIN {X 0,Y 145.091,Z 1002.94,A -85,B 0,C 180,E1 1792.898,E2 1792.898} C_VEL
LIN {X 0,Y 129.48,Z 1013.624,A -85,B 0,C 180,E1 1790.668,E2 1790.668} C_VEL
LIN {X 0,Y 113.641,Z 1022.596,A -85,B 0,C 180,E1 1787.581,E2 1787.581} C_VEL
LIN {X 0,Y 97.23,Z 1030.171,A -85,B 0,C 180,E1 1783.005,E2 1783.005} C_VEL
LIN {X 0,Y 81.806,Z 1035.835,A -85,B 0,C 180,E1 1776.44,E2 1776.44} C_VEL
LIN {X 0,Y 67.386,Z 1039.964,A -85,B 0,C 180,E1 1766.189,E2 1766.189} C_VEL
LIN {X 0,Y 55.9,Z 1042.389,A -85,B 0,C 180,E1 1750.081,E2 1750.081} C_VEL
LIN {X 0,Y 50.774,Z 1042.889,A -85,B 0,C 180,E1 1729.057,E2 1729.057} C_VEL
LIN {X 0,Y 52.115,Z 1041.788,A -85,B 0,C 180,E1 1710.272,E2 1710.272} C_VEL
LIN {X 0,Y 51.039,Z 1039.532,A -85,B 0,C 180,E1 1698.409,E2 1698.409} C_VEL
LIN {X 0,Y 50.248,Z 1038.177,A -85,B 0,C 180,E1 1692.749,E2 1692.749} C_VEL
LIN {X 0,Y 47.031,Z 1033.488,A -85,B 0,C 180,E1 1676.994,E2 1676.994} C_VEL
LIN {X 0,Y 48.077,Z 1031.863,A -85,B 0,C 180,E1 1672.098,E2 1672.098} C_VEL
LIN {X 0,Y 53.059,Z 1028.403,A -85,B 0,C 180,E1 1663.091,E2 1663.091} C_VEL
LIN {X 0,Y 67.026,Z 1030.348,A -85,B 0,C 180,E1 1646.48,E2 1646.48} C_VEL
LIN {X 0,Y 67.33,Z 1030.339,A -85,B 0,C 180,E1 1646.135,E2 1646.135} C_VEL
LIN {X 0,Y 55.64,Z 1023.763,A -85,B 0,C 180,E1 1634.569,E2 1634.569} C_VEL
LIN {X 0,Y 47.467,Z 1015.8,A -85,B 0,C 180,E1 1618.636,E2 1618.636} C_VEL
LIN {X 0,Y 45.6,Z 1015.272,A -85,B 0,C 180,E1 1608.616,E2 1608.616} C_VEL
LIN {X 0,Y 46.09,Z 1014.285,A -85,B 0,C 180,E1 1590.066,E2 1590.066} C_VEL
LIN {X 0,Y 60.524,Z 1012.005,A -85,B 0,C 180,E1 1559.576,E2 1559.576} C_VEL
LIN {X 0,Y 51.002,Z 1019.248,A -85,B 0,C 180,E1 1544.768,E2 1544.768} C_VEL
LIN {X 0,Y 45.574,Z 1024.693,A -85,B 0,C 180,E1 1524.969,E2 1524.969} C_VEL
LIN {X 0,Y 45.855,Z 1028.422,A -85,B 0,C 180,E1 1502.752,E2 1502.752} C_VEL
LIN {X 0,Y 51.98,Z 1030.449,A -85,B 0,C 180,E1 1483.038,E2 1483.038} C_VEL
LIN {X 0,Y 62.512,Z 1030.806,A -85,B 0,C 180,E1 1468.399,E2 1468.399} C_VEL
LIN {X 0,Y 76.632,Z 1029.331,A -85,B 0,C 180,E1 1457.742,E2 1457.742} C_VEL
LIN {X 0,Y 92.007,Z 1026.024,A -85,B 0,C 180,E1 1450.647,E2 1450.647} C_VEL
LIN {X 0,Y 107.53,Z 1021.018,A -85,B 0,C 180,E1 1445.782,E2 1445.782} C_VEL
LIN {X 0,Y 123.072,Z 1014.245,A -85,B 0,C 180,E1 1442.216,E2 1442.216} C_VEL
LIN {X 0,Y 137.982,Z 1005.988,A -85,B 0,C 180,E1 1439.569,E2 1439.569} C_VEL
LIN {X 0,Y 152.117,Z 996.317,A -85,B 0,C 180,E1 1437.535,E2 1437.535} C_VEL
LIN {X 0,Y 155.427,Z 993.81,A -85,B 0,C 180,E1 1437.081,E2 1437.081} C_VEL
LIN {X 0,Y 140.375,Z 1005.309,A -85,B 0,C 180,E1 1435.691,E2 1435.691} C_VEL
LIN {X 0,Y 124.723,Z 1015.179,A -85,B 0,C 180,E1 1433.744,E2 1433.744} C_VEL
LIN {X 0,Y 108.343,Z 1023.635,A -85,B 0,C 180,E1 1430.911,E2 1430.911} C_VEL
LIN {X 0,Y 91.462,Z 1030.644,A -85,B 0,C 180,E1 1426.635,E2 1426.635} C_VEL
LIN {X 0,Y 75.416,Z 1035.835,A -85,B 0,C 180,E1 1420.268,E2 1420.268} C_VEL
LIN {X 0,Y 60.179,Z 1039.51,A -85,B 0,C 180,E1 1409.761,E2 1409.761} C_VEL
LIN {X 0,Y 48.368,Z 1041.37,A -85,B 0,C 180,E1 1393.009,E2 1393.009} C_VEL
LIN {X 0,Y 42.877,Z 1041.457,A -85,B 0,C 180,E1 1369.051,E2 1369.051} C_VEL
LIN {X 0,Y 43.992,Z 1040.334,A -85,B 0,C 180,E1 1349.938,E2 1349.938} C_VEL
LIN {X 0,Y 43.916,Z 1036.153,A -85,B 0,C 180,E1 1327.225,E2 1327.225} C_VEL
LIN {X 0,Y 48.077,Z 1031.863,A -85,B 0,C 180,E1 1312.098,E2 1312.098} C_VEL
LIN {X 0,Y 49.648,Z 1030.026,A -85,B 0,C 180,E1 1306.583,E2 1306.583} C_VEL
LIN {X 0,Y 51.074,Z 1027.504,A -85,B 0,C 180,E1 1296.601,E2 1296.601} C_VEL
LIN {X 0,Y 53.467,Z 1026.726,A -85,B 0,C 180,E1 1289.596,E2 1289.596} C_VEL
LIN {X 0,Y 55.343,Z 1026.859,A -85,B 0,C 180,E1 1287.109,E2 1287.109} C_VEL
LIN {X 0,Y 55.723,Z 1026.897,A -85,B 0,C 180,E1 1286.651,E2 1286.651} C_VEL
LIN {X 0,Y 45.56,Z 1020.385,A -85,B 0,C 180,E1 1274.504,E2 1274.504} C_VEL
LIN {X 0,Y 41.053,Z 1019.632,A -85,B 0,C 180,E1 1262.99,E2 1262.99} C_VEL
LIN {X 0,Y 38.426,Z 1018.764,A -85,B 0,C 180,E1 1247.219,E2 1247.219} C_VEL
LIN {X 0,Y 50.467,Z 1016.033,A -85,B 0,C 180,E1 1200.02,E2 1200.02} C_VEL
LIN {X 0,Y 41.318,Z 1022.364,A -85,B 0,C 180,E1 1182.583,E2 1182.583} C_VEL
LIN {X 0,Y 37.017,Z 1027.38,A -85,B 0,C 180,E1 1156.52,E2 1156.52} C_VEL
LIN {X 0,Y 40.434,Z 1030.565,A -85,B 0,C 180,E1 1129.994,E2 1129.994} C_VEL
LIN {X 0,Y 49.975,Z 1032.016,A -85,B 0,C 180,E1 1110.655,E2 1110.655} C_VEL
LIN {X 0,Y 63.959,Z 1031.679,A -85,B 0,C 180,E1 1097.53,E2 1097.53} C_VEL
LIN {X 0,Y 79.549,Z 1029.503,A -85,B 0,C 180,E1 1089.406,E2 1089.406} C_VEL
LIN {X 0,Y 95.238,Z 1025.699,A -85,B 0,C 180,E1 1084.184,E2 1084.184} C_VEL
LIN {X 0,Y 110.986,Z 1020.256,A -85,B 0,C 180,E1 1080.504,E2 1080.504} C_VEL
LIN {X 0,Y 126.642,Z 1013.13,A -85,B 0,C 180,E1 1077.767,E2 1077.767} C_VEL
LIN {X 0,Y 110.294,Z 1021.547,A -85,B 0,C 180,E1 1075.686,E2 1075.686} C_VEL
LIN {X 0,Y 92.796,Z 1028.717,A -85,B 0,C 180,E1 1072.419,E2 1072.419} C_VEL
LIN {X 0,Y 74.884,Z 1034.322,A -85,B 0,C 180,E1 1067.077,E2 1067.077} C_VEL
LIN {X 0,Y 58.137,Z 1038.07,A -85,B 0,C 180,E1 1058.228,E2 1058.228} C_VEL
LIN {X 0,Y 43.967,Z 1040.028,A -85,B 0,C 180,E1 1042.738,E2 1042.738} C_VEL
LIN {X 0,Y 35.515,Z 1040.161,A -85,B 0,C 180,E1 1015.729,E2 1015.729} C_VEL
LIN {X 0,Y 35.92,Z 1038.925,A -85,B 0,C 180,E1 989.996,E2 989.996} C_VEL
LIN {X 0,Y 36.578,Z 1034.576,A -85,B 0,C 180,E1 962.305,E2 962.305} C_VEL
LIN {X 0,Y 45.352,Z 1028.024,A -85,B 0,C 180,E1 939.494,E2 939.494} C_VEL
LIN {X 0,Y 49.333,Z 1025.812,A -85,B 0,C 180,E1 934.437,E2 934.437} C_VEL
LIN {X 0,Y 55.343,Z 1026.859,A -85,B 0,C 180,E1 927.109,E2 927.109} C_VEL
LIN {X 0,Y 54.651,Z 1027.472,A -85,B 0,C 180,E1 926.54,E2 926.54} C_VEL
LIN {X 0,Y 51.085,Z 1028.61,A -85,B 0,C 180,E1 927.205,E2 927.205} C_VEL
LIN {X 0,Y 44.894,Z 1029.802,A -85,B 0,C 180,E1 930.625,E2 930.625} C_VEL
LIN {X 0,Y 32.514,Z 1031.993,A -85,B 0,C 180,E1 946.547,E2 946.547} C_VEL
LIN {X 0,Y 28.72,Z 1033.778,A -85,B 0,C 180,E1 959.758,E2 959.758} C_VEL
LIN {X 0,Y 27.878,Z 1037.562,A -85,B 0,C 180,E1 991.022,E2 991.022} C_VEL
LIN {X 0,Y 29.704,Z 1038.961,A -85,B 0,C 180,E1 1029.753,E2 1029.753} C_VEL
LIN {X 0,Y 41.869,Z 1038.59,A -85,B 0,C 180,E1 1055.148,E2 1055.148} C_VEL
LIN {X 0,Y 58.358,Z 1036.466,A -85,B 0,C 180,E1 1067.565,E2 1067.565} C_VEL
LIN {X 0,Y 77.357,Z 1032.317,A -85,B 0,C 180,E1 1074.395,E2 1074.395} C_VEL
LIN {X 0,Y 95.044,Z 1026.807,A -85,B 0,C 180,E1 1077.972,E2 1077.972} C_VEL
LIN {X 0,Y 98.271,Z 1025.617,A -85,B 0,C 180,E1 1078.481,E2 1078.481} C_VEL
LIN {X 0,Y 81.072,Z 1030.063,A -85,B 0,C 180,E1 1082.639,E2 1082.639} C_VEL
LIN {X 0,Y 64.31,Z 1032.586,A -85,B 0,C 180,E1 1088.946,E2 1088.946} C_VEL
LIN {X 0,Y 48.731,Z 1033.295,A -85,B 0,C 180,E1 1099.303,E2 1099.303} C_VEL
LIN {X 0,Y 35.713,Z 1032.195,A -85,B 0,C 180,E1 1118.023,E2 1118.023} C_VEL
LIN {X 0,Y 29.27,Z 1029.433,A -85,B 0,C 180,E1 1147.934,E2 1147.934} C_VEL
LIN {X 0,Y 32.061,Z 1024.989,A -85,B 0,C 180,E1 1180.789,E2 1180.789} C_VEL
LIN {X 0,Y 40.294,Z 1019.754,A -85,B 0,C 180,E1 1201.114,E2 1201.114} C_VEL
LIN {X 0,Y 35.496,Z 1023.369,A -85,B 0,C 180,E1 1271.369,E2 1271.369} C_VEL
LIN {X 0,Y 44.049,Z 1024.441,A -85,B 0,C 180,E1 1287.161,E2 1287.161} C_VEL
LIN {X 0,Y 32.009,Z 1031.337,A -85,B 0,C 180,E1 1306.584,E2 1306.584} C_VEL
LIN {X 0,Y 28.72,Z 1033.778,A -85,B 0,C 180,E1 1319.758,E2 1319.758} C_VEL
LIN {X 0,Y 26.509,Z 1034.967,A -85,B 0,C 180,E1 1329.06,E2 1329.06} C_VEL
LIN {X 0,Y 22.849,Z 1035.906,A -85,B 0,C 180,E1 1342.03,E2 1342.03} C_VEL
LIN {X 0,Y 19.4,Z 1036.852,A -85,B 0,C 180,E1 1372.712,E2 1372.712} C_VEL
LIN {X 0,Y 19.501,Z 1036.919,A -85,B 0,C 180,E1 1374.976,E2 1374.976} C_VEL
LIN {X 0,Y 29.714,Z 1037.699,A -85,B 0,C 180,E1 1415.292,E2 1415.292} C_VEL
LIN {X 0,Y 46.556,Z 1036.744,A -85,B 0,C 180,E1 1431.065,E2 1431.065} C_VEL
LIN {X 0,Y 65.029,Z 1034.007,A -85,B 0,C 180,E1 1437.977,E2 1437.977} C_VEL
LIN {X 0,Y 70.458,Z 1032.858,A -85,B 0,C 180,E1 1439.323,E2 1439.323} C_VEL
LIN {X 0,Y 53.258,Z 1034.406,A -85,B 0,C 180,E1 1445.75,E2 1445.75} C_VEL
LIN {X 0,Y 36.819,Z 1034.144,A -85,B 0,C 180,E1 1458.124,E2 1458.124} C_VEL
LIN {X 0,Y 24.345,Z 1032.107,A -85,B 0,C 180,E1 1484.289,E2 1484.289} C_VEL
LIN {X 0,Y 21.848,Z 1028.297,A -85,B 0,C 180,E1 1530.007,E2 1530.007} C_VEL
LIN {X 0,Y 30.024,Z 1023.292,A -85,B 0,C 180,E1 1562.049,E2 1562.049} C_VEL
LIN {X 0,Y 29.767,Z 1026.621,A -85,B 0,C 180,E1 1639.623,E2 1639.623} C_VEL
LIN {X 0,Y 32.339,Z 1026.982,A -85,B 0,C 180,E1 1645.231,E2 1645.231} C_VEL
LIN {X 0,Y 20.993,Z 1032.93,A -85,B 0,C 180,E1 1675.133,E2 1675.133} C_VEL
LIN {X 0,Y 19.796,Z 1036.087,A -85,B 0,C 180,E1 1711.439,E2 1711.439} C_VEL
LIN {X 0,Y 19.501,Z 1036.919,A -85,B 0,C 180,E1 1734.976,E2 1734.976} C_VEL
LIN {X 0,Y 21.254,Z 1037.33,A -85,B 0,C 180,E1 1756.358,E2 1756.358} C_VEL
LIN {X 0,Y 32.993,Z 1036.546,A -85,B 0,C 180,E1 1793.925,E2 1793.925} C_VEL
LIN {X 0,Y 39.491,Z 1036.041,A -85,B 0,C 180,E1 1798.885,E2 1798.885} C_VEL
LIN {X 0,Y 43.353,Z 1035.734,A -85,B 0,C 180,E1 1800.394,E2 1800.394} C_VEL
LIN {X 0,Y 26.687,Z 1034.663,A -85,B 0,C 180,E1 1813.091,E2 1813.091} C_VEL
LIN {X 0,Y 14.362,Z 1031.955,A -85,B 0,C 180,E1 1851.215,E2 1851.215} C_VEL
LIN {X 0,Y 17.58,Z 1027.591,A -85,B 0,C 180,E1 1917.074,E2 1917.074} C_VEL
LIN {X 0,Y 19.66,Z 1026.597,A -85,B 0,C 180,E1 1924.382,E2 1924.382} C_VEL
LIN {X 0,Y 20.808,Z 1029.001,A -85,B 0,C 180,E1 2001.43,E2 2001.43} C_VEL
LIN {X 0,Y 11.407,Z 1034.053,A -85,B 0,C 180,E1 2059.89,E2 2059.89} C_VEL
LIN {X 0,Y 11.6,Z 1034.681,A -85,B 0,C 180,E1 2074.932,E2 2074.932} C_VEL
LIN {X 0,Y 20.934,Z 1036.272,A -85,B 0,C 180,E1 2142.77,E2 2142.77} C_VEL
LIN {X 0,Y 39.491,Z 1036.041,A -85,B 0,C 180,E1 2158.885,E2 2158.885} C_VEL
LIN {X 0,Y 38.6,Z 1035.9,A -85,B 0,C 180,E1 2160.345,E2 2160.345} C_VEL
LIN {X 0,Y 32.151,Z 1035.66,A -85,B 0,C 180,E1 2162.888,E2 2162.888} C_VEL
LIN {X 0,Y 14.105,Z 1034.162,A -85,B 0,C 180,E1 2170.632,E2 2170.632} C_VEL
LIN {X 0,Y 6.046,Z 1032.398,A -85,B 0,C 180,E1 2205.029,E2 2205.029} C_VEL
LIN {X 0,Y 9.396,Z 1029.668,A -85,B 0,C 180,E1 2291.833,E2 2291.833} C_VEL
LIN {X 0,Y 9.282,Z 1030.645,A -85,B 0,C 180,E1 2350.032,E2 2350.032} C_VEL
LIN {X 0,Y 3.627,Z 1033.134,A -85,B 0,C 180,E1 2437.88,E2 2437.88} C_VEL
LIN {X 0,Y 16.018,Z 1034.692,A -85,B 0,C 180,E1 2523.062,E2 2523.062} C_VEL
LIN {X 0,Y 6.046,Z 1032.398,A -85,B 0,C 180,E1 2565.029,E2 2565.029} C_VEL
LIN {X 0,Y 5.288,Z 1034.347,A -85,B 0,C 180,E1 2588.821,E2 2588.821} C_VEL
LIN {X 0,Y 5.288,Z 1116.5,A -85,B 0,C 180,E1 2588.821,E2 2588.821} C_VEL
LIN {X 0,Y 5.288,Z 1116.5,A -85,B 0,C 180,E1 2588.821,E2 2588.821}

QRS_NEXT_CUT()

QRS_NEXT()
QRS_HOME()

END
